{attribute 'TcGenerated'}
{attribute 'no-analysis'}
{attribute 'linkalways'}
// This function has been automatically generated from the project information.
VAR_GLOBAL CONSTANT
	{attribute 'const_non_replaced'}
	stLibVersion_TwinCAT_Open_Framework_Core : ST_LibVersion := (iMajor := 1, iMinor := 0, iBuild := 13, iRevision := 0, nFlags := 0, sVersion := '1.0.13.0');
END_VAR

(* stored: Version 1.1.0.1
   GVL Global_Version: Id {17c7f750-d944-4f9a-bd27-86ab7ab11e77} *)
